{attribute 'GeneratedUsingTerminal: EL6201-0000-0017'}
{attribute addProperty BoxType "EL6201-0000-0017"}
{attribute addProperty Id "Slave_1A_DI0BOOL1Slave_1A_DI1BOOL1Slave_1A_DI2BOOL1Slave_1A_DI3BOOL1Slave_1B_DI0BOOL1Slave_1B_DI1BOOL1Slave_1B_DI2BOOL1Slave_1B_DI3BOOL1"}
{attribute addProperty CRC "741365928"}
{attribute addProperty Size "8"}
TYPE Slave_1_Inputs_2C3058A8 :
STRUCT
	{attribute addProperty Name "Slave_1A_DI0"}
	Slave_1A_DI0 : BOOL;
	{attribute addProperty Name "Slave_1A_DI1"}
	Slave_1A_DI1 : BOOL;
	{attribute addProperty Name "Slave_1A_DI2"}
	Slave_1A_DI2 : BOOL;
	{attribute addProperty Name "Slave_1A_DI3"}
	Slave_1A_DI3 : BOOL;
	{attribute addProperty Name "Slave_1B_DI0"}
	Slave_1B_DI0 : BOOL;
	{attribute addProperty Name "Slave_1B_DI1"}
	Slave_1B_DI1 : BOOL;
	{attribute addProperty Name "Slave_1B_DI2"}
	Slave_1B_DI2 : BOOL;
	{attribute addProperty Name "Slave_1B_DI3"}
	Slave_1B_DI3 : BOOL;
END_STRUCT
END_TYPE

(* stored: Version 1.2.0.0, ProductVersion 3.1.4024.9
   DUT Slave_1_Inputs_2C3058A8: Id {27223d68-c3bd-47c1-94a9-e82eb2d1e39d} *)
